// TIA Portal V18 export
FUNCTION "SS1_774A1_16DO_IO_Update" : Void   // FC11070, LAD
{ S7_Optimized_Access := 'TRUE' }
VERSION : 0.1
// stored: AutoNumber false, IsIECCheckEnabled false, SetENOAutomatically false, UDAEnableTagReadback false
BEGIN

REGION Network 1: DQa0
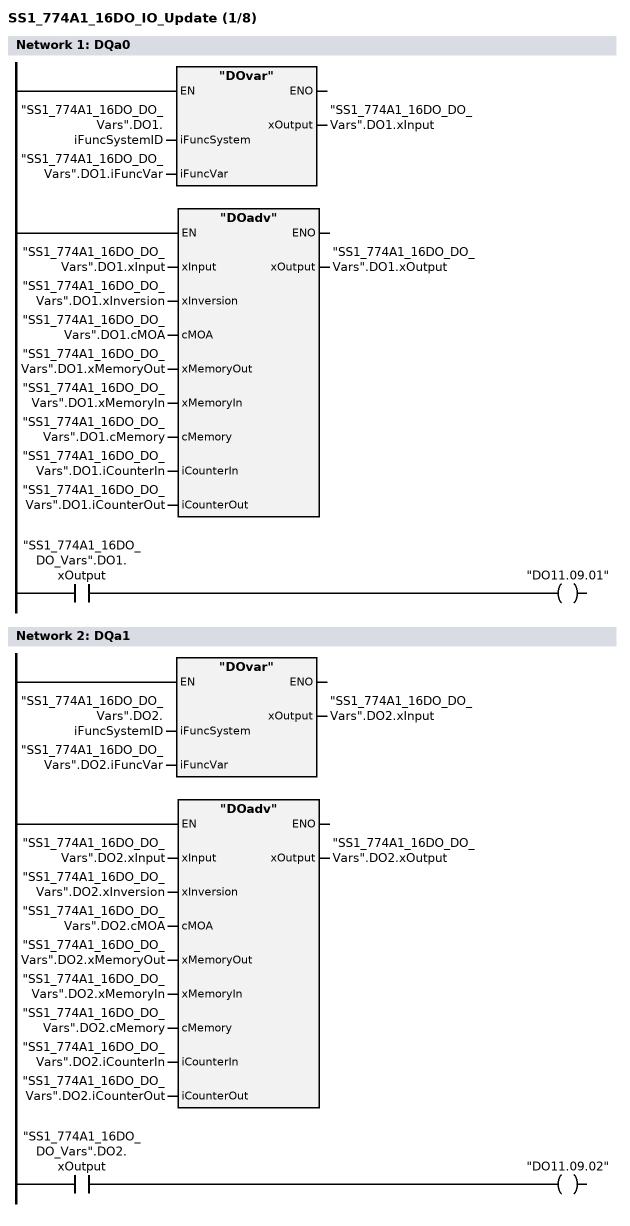
   RUNG wire#powerrail
      "DOvar"(iFuncSystem := "SS1_774A1_16DO_DO_Vars".DO1.iFuncSystemID, iFuncVar := "SS1_774A1_16DO_DO_Vars".DO1.iFuncVar, xOutput => "SS1_774A1_16DO_DO_Vars".DO1.xInput)
   END_RUNG
   RUNG wire#powerrail
      "DOadv"(xInput := "SS1_774A1_16DO_DO_Vars".DO1.xInput, xInversion := "SS1_774A1_16DO_DO_Vars".DO1.xInversion, cMOA := "SS1_774A1_16DO_DO_Vars".DO1.cMOA, xMemoryOut := "SS1_774A1_16DO_DO_Vars".DO1.xMemoryOut, xMemoryIn := "SS1_774A1_16DO_DO_Vars".DO1.xMemoryIn, cMemory := "SS1_774A1_16DO_DO_Vars".DO1.cMemory, iCounterIn := "SS1_774A1_16DO_DO_Vars".DO1.iCounterIn, iCounterOut := "SS1_774A1_16DO_DO_Vars".DO1.iCounterOut, xOutput => "SS1_774A1_16DO_DO_Vars".DO1.xOutput)
   END_RUNG
   RUNG wire#powerrail
      Contact( "SS1_774A1_16DO_DO_Vars".DO1.xOutput )
      Coil( "DO11.09.01" )
   END_RUNG
   // the same network as SCL:
   "DOvar"(iFuncSystem := "SS1_774A1_16DO_DO_Vars".DO1.iFuncSystemID,
           iFuncVar := "SS1_774A1_16DO_DO_Vars".DO1.iFuncVar,
           xOutput => "SS1_774A1_16DO_DO_Vars".DO1.xInput);
   "DOadv"(xInput := "SS1_774A1_16DO_DO_Vars".DO1.xInput,
           xInversion := "SS1_774A1_16DO_DO_Vars".DO1.xInversion,
           cMOA := "SS1_774A1_16DO_DO_Vars".DO1.cMOA,
           xMemoryOut := "SS1_774A1_16DO_DO_Vars".DO1.xMemoryOut,
           xMemoryIn := "SS1_774A1_16DO_DO_Vars".DO1.xMemoryIn,
           cMemory := "SS1_774A1_16DO_DO_Vars".DO1.cMemory,
           iCounterIn := "SS1_774A1_16DO_DO_Vars".DO1.iCounterIn,
           iCounterOut := "SS1_774A1_16DO_DO_Vars".DO1.iCounterOut,
           xOutput => "SS1_774A1_16DO_DO_Vars".DO1.xOutput);
   "DO11.09.01" := "SS1_774A1_16DO_DO_Vars".DO1.xOutput;
END_REGION

REGION Network 2: DQa1
   RUNG wire#powerrail
      "DOvar"(iFuncSystem := "SS1_774A1_16DO_DO_Vars".DO2.iFuncSystemID, iFuncVar := "SS1_774A1_16DO_DO_Vars".DO2.iFuncVar, xOutput => "SS1_774A1_16DO_DO_Vars".DO2.xInput)
   END_RUNG
   RUNG wire#powerrail
      "DOadv"(xInput := "SS1_774A1_16DO_DO_Vars".DO2.xInput, xInversion := "SS1_774A1_16DO_DO_Vars".DO2.xInversion, cMOA := "SS1_774A1_16DO_DO_Vars".DO2.cMOA, xMemoryOut := "SS1_774A1_16DO_DO_Vars".DO2.xMemoryOut, xMemoryIn := "SS1_774A1_16DO_DO_Vars".DO2.xMemoryIn, cMemory := "SS1_774A1_16DO_DO_Vars".DO2.cMemory, iCounterIn := "SS1_774A1_16DO_DO_Vars".DO2.iCounterIn, iCounterOut := "SS1_774A1_16DO_DO_Vars".DO2.iCounterOut, xOutput => "SS1_774A1_16DO_DO_Vars".DO2.xOutput)
   END_RUNG
   RUNG wire#powerrail
      Contact( "SS1_774A1_16DO_DO_Vars".DO2.xOutput )
      Coil( "DO11.09.02" )
   END_RUNG
   // the same network as SCL:
   "DOvar"(iFuncSystem := "SS1_774A1_16DO_DO_Vars".DO2.iFuncSystemID,
           iFuncVar := "SS1_774A1_16DO_DO_Vars".DO2.iFuncVar,
           xOutput => "SS1_774A1_16DO_DO_Vars".DO2.xInput);
   "DOadv"(xInput := "SS1_774A1_16DO_DO_Vars".DO2.xInput,
           xInversion := "SS1_774A1_16DO_DO_Vars".DO2.xInversion,
           cMOA := "SS1_774A1_16DO_DO_Vars".DO2.cMOA,
           xMemoryOut := "SS1_774A1_16DO_DO_Vars".DO2.xMemoryOut,
           xMemoryIn := "SS1_774A1_16DO_DO_Vars".DO2.xMemoryIn,
           cMemory := "SS1_774A1_16DO_DO_Vars".DO2.cMemory,
           iCounterIn := "SS1_774A1_16DO_DO_Vars".DO2.iCounterIn,
           iCounterOut := "SS1_774A1_16DO_DO_Vars".DO2.iCounterOut,
           xOutput => "SS1_774A1_16DO_DO_Vars".DO2.xOutput);
   "DO11.09.02" := "SS1_774A1_16DO_DO_Vars".DO2.xOutput;
END_REGION

REGION Network 3: DQa2
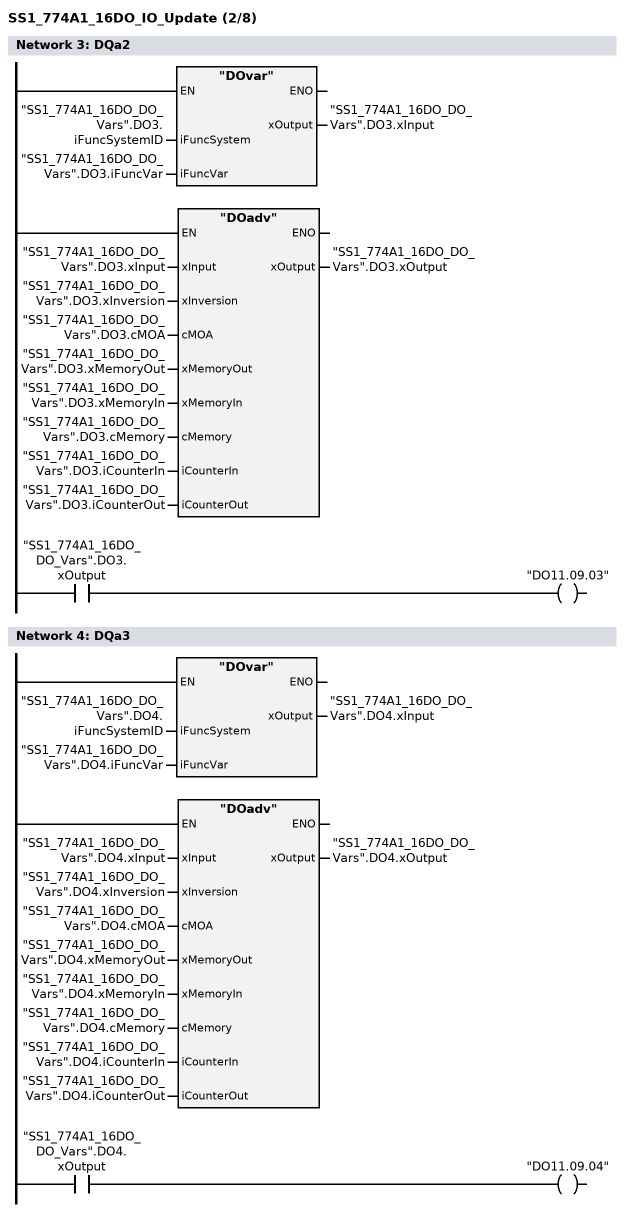
   RUNG wire#powerrail
      "DOvar"(iFuncSystem := "SS1_774A1_16DO_DO_Vars".DO3.iFuncSystemID, iFuncVar := "SS1_774A1_16DO_DO_Vars".DO3.iFuncVar, xOutput => "SS1_774A1_16DO_DO_Vars".DO3.xInput)
   END_RUNG
   RUNG wire#powerrail
      "DOadv"(xInput := "SS1_774A1_16DO_DO_Vars".DO3.xInput, xInversion := "SS1_774A1_16DO_DO_Vars".DO3.xInversion, cMOA := "SS1_774A1_16DO_DO_Vars".DO3.cMOA, xMemoryOut := "SS1_774A1_16DO_DO_Vars".DO3.xMemoryOut, xMemoryIn := "SS1_774A1_16DO_DO_Vars".DO3.xMemoryIn, cMemory := "SS1_774A1_16DO_DO_Vars".DO3.cMemory, iCounterIn := "SS1_774A1_16DO_DO_Vars".DO3.iCounterIn, iCounterOut := "SS1_774A1_16DO_DO_Vars".DO3.iCounterOut, xOutput => "SS1_774A1_16DO_DO_Vars".DO3.xOutput)
   END_RUNG
   RUNG wire#powerrail
      Contact( "SS1_774A1_16DO_DO_Vars".DO3.xOutput )
      Coil( "DO11.09.03" )
   END_RUNG
   // the same network as SCL:
   "DOvar"(iFuncSystem := "SS1_774A1_16DO_DO_Vars".DO3.iFuncSystemID,
           iFuncVar := "SS1_774A1_16DO_DO_Vars".DO3.iFuncVar,
           xOutput => "SS1_774A1_16DO_DO_Vars".DO3.xInput);
   "DOadv"(xInput := "SS1_774A1_16DO_DO_Vars".DO3.xInput,
           xInversion := "SS1_774A1_16DO_DO_Vars".DO3.xInversion,
           cMOA := "SS1_774A1_16DO_DO_Vars".DO3.cMOA,
           xMemoryOut := "SS1_774A1_16DO_DO_Vars".DO3.xMemoryOut,
           xMemoryIn := "SS1_774A1_16DO_DO_Vars".DO3.xMemoryIn,
           cMemory := "SS1_774A1_16DO_DO_Vars".DO3.cMemory,
           iCounterIn := "SS1_774A1_16DO_DO_Vars".DO3.iCounterIn,
           iCounterOut := "SS1_774A1_16DO_DO_Vars".DO3.iCounterOut,
           xOutput => "SS1_774A1_16DO_DO_Vars".DO3.xOutput);
   "DO11.09.03" := "SS1_774A1_16DO_DO_Vars".DO3.xOutput;
END_REGION

REGION Network 4: DQa3
   RUNG wire#powerrail
      "DOvar"(iFuncSystem := "SS1_774A1_16DO_DO_Vars".DO4.iFuncSystemID, iFuncVar := "SS1_774A1_16DO_DO_Vars".DO4.iFuncVar, xOutput => "SS1_774A1_16DO_DO_Vars".DO4.xInput)
   END_RUNG
   RUNG wire#powerrail
      "DOadv"(xInput := "SS1_774A1_16DO_DO_Vars".DO4.xInput, xInversion := "SS1_774A1_16DO_DO_Vars".DO4.xInversion, cMOA := "SS1_774A1_16DO_DO_Vars".DO4.cMOA, xMemoryOut := "SS1_774A1_16DO_DO_Vars".DO4.xMemoryOut, xMemoryIn := "SS1_774A1_16DO_DO_Vars".DO4.xMemoryIn, cMemory := "SS1_774A1_16DO_DO_Vars".DO4.cMemory, iCounterIn := "SS1_774A1_16DO_DO_Vars".DO4.iCounterIn, iCounterOut := "SS1_774A1_16DO_DO_Vars".DO4.iCounterOut, xOutput => "SS1_774A1_16DO_DO_Vars".DO4.xOutput)
   END_RUNG
   RUNG wire#powerrail
      Contact( "SS1_774A1_16DO_DO_Vars".DO4.xOutput )
      Coil( "DO11.09.04" )
   END_RUNG
   // the same network as SCL:
   "DOvar"(iFuncSystem := "SS1_774A1_16DO_DO_Vars".DO4.iFuncSystemID,
           iFuncVar := "SS1_774A1_16DO_DO_Vars".DO4.iFuncVar,
           xOutput => "SS1_774A1_16DO_DO_Vars".DO4.xInput);
   "DOadv"(xInput := "SS1_774A1_16DO_DO_Vars".DO4.xInput,
           xInversion := "SS1_774A1_16DO_DO_Vars".DO4.xInversion,
           cMOA := "SS1_774A1_16DO_DO_Vars".DO4.cMOA,
           xMemoryOut := "SS1_774A1_16DO_DO_Vars".DO4.xMemoryOut,
           xMemoryIn := "SS1_774A1_16DO_DO_Vars".DO4.xMemoryIn,
           cMemory := "SS1_774A1_16DO_DO_Vars".DO4.cMemory,
           iCounterIn := "SS1_774A1_16DO_DO_Vars".DO4.iCounterIn,
           iCounterOut := "SS1_774A1_16DO_DO_Vars".DO4.iCounterOut,
           xOutput => "SS1_774A1_16DO_DO_Vars".DO4.xOutput);
   "DO11.09.04" := "SS1_774A1_16DO_DO_Vars".DO4.xOutput;
END_REGION

REGION Network 5: DQa4
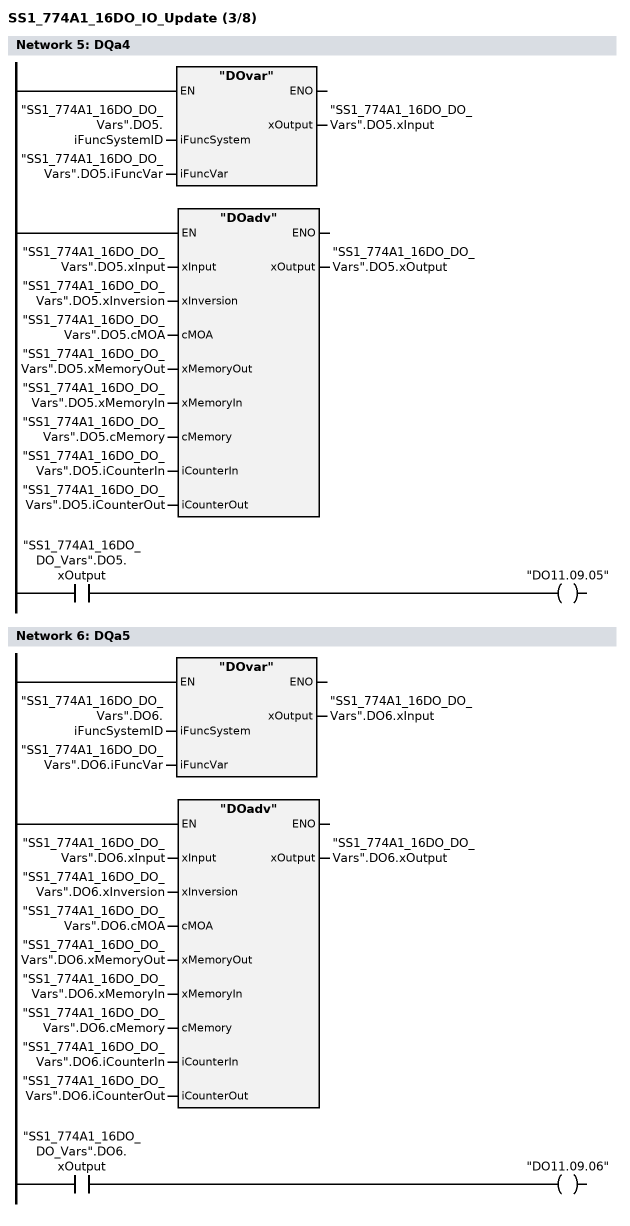
   RUNG wire#powerrail
      "DOvar"(iFuncSystem := "SS1_774A1_16DO_DO_Vars".DO5.iFuncSystemID, iFuncVar := "SS1_774A1_16DO_DO_Vars".DO5.iFuncVar, xOutput => "SS1_774A1_16DO_DO_Vars".DO5.xInput)
   END_RUNG
   RUNG wire#powerrail
      "DOadv"(xInput := "SS1_774A1_16DO_DO_Vars".DO5.xInput, xInversion := "SS1_774A1_16DO_DO_Vars".DO5.xInversion, cMOA := "SS1_774A1_16DO_DO_Vars".DO5.cMOA, xMemoryOut := "SS1_774A1_16DO_DO_Vars".DO5.xMemoryOut, xMemoryIn := "SS1_774A1_16DO_DO_Vars".DO5.xMemoryIn, cMemory := "SS1_774A1_16DO_DO_Vars".DO5.cMemory, iCounterIn := "SS1_774A1_16DO_DO_Vars".DO5.iCounterIn, iCounterOut := "SS1_774A1_16DO_DO_Vars".DO5.iCounterOut, xOutput => "SS1_774A1_16DO_DO_Vars".DO5.xOutput)
   END_RUNG
   RUNG wire#powerrail
      Contact( "SS1_774A1_16DO_DO_Vars".DO5.xOutput )
      Coil( "DO11.09.05" )
   END_RUNG
   // the same network as SCL:
   "DOvar"(iFuncSystem := "SS1_774A1_16DO_DO_Vars".DO5.iFuncSystemID,
           iFuncVar := "SS1_774A1_16DO_DO_Vars".DO5.iFuncVar,
           xOutput => "SS1_774A1_16DO_DO_Vars".DO5.xInput);
   "DOadv"(xInput := "SS1_774A1_16DO_DO_Vars".DO5.xInput,
           xInversion := "SS1_774A1_16DO_DO_Vars".DO5.xInversion,
           cMOA := "SS1_774A1_16DO_DO_Vars".DO5.cMOA,
           xMemoryOut := "SS1_774A1_16DO_DO_Vars".DO5.xMemoryOut,
           xMemoryIn := "SS1_774A1_16DO_DO_Vars".DO5.xMemoryIn,
           cMemory := "SS1_774A1_16DO_DO_Vars".DO5.cMemory,
           iCounterIn := "SS1_774A1_16DO_DO_Vars".DO5.iCounterIn,
           iCounterOut := "SS1_774A1_16DO_DO_Vars".DO5.iCounterOut,
           xOutput => "SS1_774A1_16DO_DO_Vars".DO5.xOutput);
   "DO11.09.05" := "SS1_774A1_16DO_DO_Vars".DO5.xOutput;
END_REGION

REGION Network 6: DQa5
   RUNG wire#powerrail
      "DOvar"(iFuncSystem := "SS1_774A1_16DO_DO_Vars".DO6.iFuncSystemID, iFuncVar := "SS1_774A1_16DO_DO_Vars".DO6.iFuncVar, xOutput => "SS1_774A1_16DO_DO_Vars".DO6.xInput)
   END_RUNG
   RUNG wire#powerrail
      "DOadv"(xInput := "SS1_774A1_16DO_DO_Vars".DO6.xInput, xInversion := "SS1_774A1_16DO_DO_Vars".DO6.xInversion, cMOA := "SS1_774A1_16DO_DO_Vars".DO6.cMOA, xMemoryOut := "SS1_774A1_16DO_DO_Vars".DO6.xMemoryOut, xMemoryIn := "SS1_774A1_16DO_DO_Vars".DO6.xMemoryIn, cMemory := "SS1_774A1_16DO_DO_Vars".DO6.cMemory, iCounterIn := "SS1_774A1_16DO_DO_Vars".DO6.iCounterIn, iCounterOut := "SS1_774A1_16DO_DO_Vars".DO6.iCounterOut, xOutput => "SS1_774A1_16DO_DO_Vars".DO6.xOutput)
   END_RUNG
   RUNG wire#powerrail
      Contact( "SS1_774A1_16DO_DO_Vars".DO6.xOutput )
      Coil( "DO11.09.06" )
   END_RUNG
   // the same network as SCL:
   "DOvar"(iFuncSystem := "SS1_774A1_16DO_DO_Vars".DO6.iFuncSystemID,
           iFuncVar := "SS1_774A1_16DO_DO_Vars".DO6.iFuncVar,
           xOutput => "SS1_774A1_16DO_DO_Vars".DO6.xInput);
   "DOadv"(xInput := "SS1_774A1_16DO_DO_Vars".DO6.xInput,
           xInversion := "SS1_774A1_16DO_DO_Vars".DO6.xInversion,
           cMOA := "SS1_774A1_16DO_DO_Vars".DO6.cMOA,
           xMemoryOut := "SS1_774A1_16DO_DO_Vars".DO6.xMemoryOut,
           xMemoryIn := "SS1_774A1_16DO_DO_Vars".DO6.xMemoryIn,
           cMemory := "SS1_774A1_16DO_DO_Vars".DO6.cMemory,
           iCounterIn := "SS1_774A1_16DO_DO_Vars".DO6.iCounterIn,
           iCounterOut := "SS1_774A1_16DO_DO_Vars".DO6.iCounterOut,
           xOutput => "SS1_774A1_16DO_DO_Vars".DO6.xOutput);
   "DO11.09.06" := "SS1_774A1_16DO_DO_Vars".DO6.xOutput;
END_REGION

REGION Network 7: DQa6
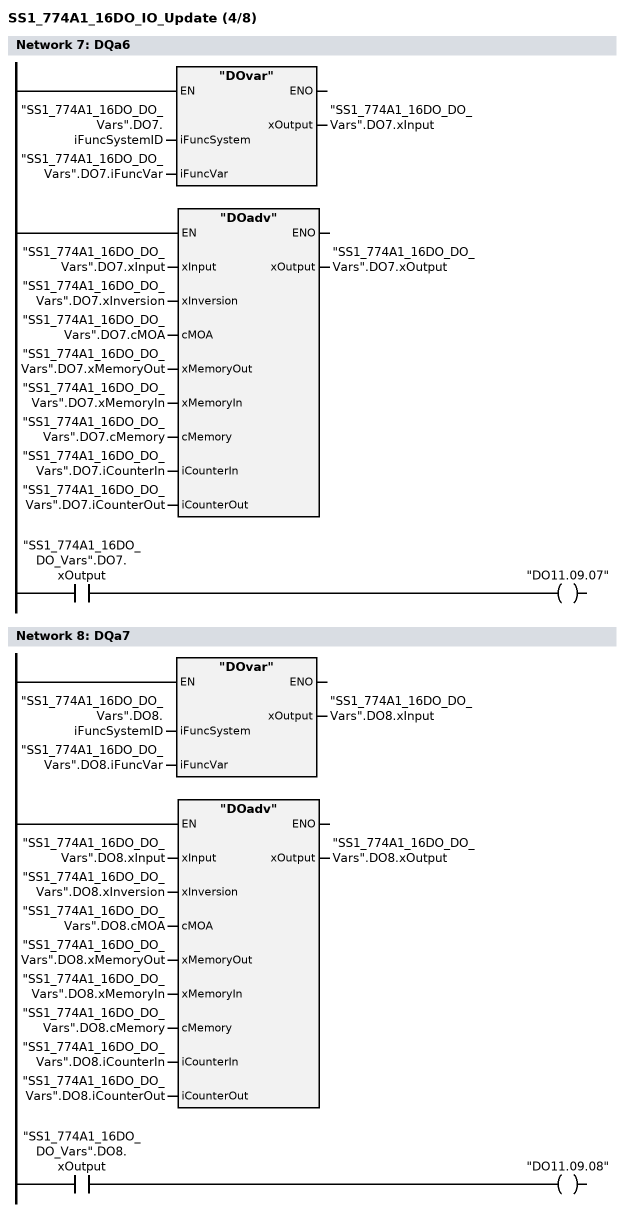
   RUNG wire#powerrail
      "DOvar"(iFuncSystem := "SS1_774A1_16DO_DO_Vars".DO7.iFuncSystemID, iFuncVar := "SS1_774A1_16DO_DO_Vars".DO7.iFuncVar, xOutput => "SS1_774A1_16DO_DO_Vars".DO7.xInput)
   END_RUNG
   RUNG wire#powerrail
      "DOadv"(xInput := "SS1_774A1_16DO_DO_Vars".DO7.xInput, xInversion := "SS1_774A1_16DO_DO_Vars".DO7.xInversion, cMOA := "SS1_774A1_16DO_DO_Vars".DO7.cMOA, xMemoryOut := "SS1_774A1_16DO_DO_Vars".DO7.xMemoryOut, xMemoryIn := "SS1_774A1_16DO_DO_Vars".DO7.xMemoryIn, cMemory := "SS1_774A1_16DO_DO_Vars".DO7.cMemory, iCounterIn := "SS1_774A1_16DO_DO_Vars".DO7.iCounterIn, iCounterOut := "SS1_774A1_16DO_DO_Vars".DO7.iCounterOut, xOutput => "SS1_774A1_16DO_DO_Vars".DO7.xOutput)
   END_RUNG
   RUNG wire#powerrail
      Contact( "SS1_774A1_16DO_DO_Vars".DO7.xOutput )
      Coil( "DO11.09.07" )
   END_RUNG
   // the same network as SCL:
   "DOvar"(iFuncSystem := "SS1_774A1_16DO_DO_Vars".DO7.iFuncSystemID,
           iFuncVar := "SS1_774A1_16DO_DO_Vars".DO7.iFuncVar,
           xOutput => "SS1_774A1_16DO_DO_Vars".DO7.xInput);
   "DOadv"(xInput := "SS1_774A1_16DO_DO_Vars".DO7.xInput,
           xInversion := "SS1_774A1_16DO_DO_Vars".DO7.xInversion,
           cMOA := "SS1_774A1_16DO_DO_Vars".DO7.cMOA,
           xMemoryOut := "SS1_774A1_16DO_DO_Vars".DO7.xMemoryOut,
           xMemoryIn := "SS1_774A1_16DO_DO_Vars".DO7.xMemoryIn,
           cMemory := "SS1_774A1_16DO_DO_Vars".DO7.cMemory,
           iCounterIn := "SS1_774A1_16DO_DO_Vars".DO7.iCounterIn,
           iCounterOut := "SS1_774A1_16DO_DO_Vars".DO7.iCounterOut,
           xOutput => "SS1_774A1_16DO_DO_Vars".DO7.xOutput);
   "DO11.09.07" := "SS1_774A1_16DO_DO_Vars".DO7.xOutput;
END_REGION

REGION Network 8: DQa7
   RUNG wire#powerrail
      "DOvar"(iFuncSystem := "SS1_774A1_16DO_DO_Vars".DO8.iFuncSystemID, iFuncVar := "SS1_774A1_16DO_DO_Vars".DO8.iFuncVar, xOutput => "SS1_774A1_16DO_DO_Vars".DO8.xInput)
   END_RUNG
   RUNG wire#powerrail
      "DOadv"(xInput := "SS1_774A1_16DO_DO_Vars".DO8.xInput, xInversion := "SS1_774A1_16DO_DO_Vars".DO8.xInversion, cMOA := "SS1_774A1_16DO_DO_Vars".DO8.cMOA, xMemoryOut := "SS1_774A1_16DO_DO_Vars".DO8.xMemoryOut, xMemoryIn := "SS1_774A1_16DO_DO_Vars".DO8.xMemoryIn, cMemory := "SS1_774A1_16DO_DO_Vars".DO8.cMemory, iCounterIn := "SS1_774A1_16DO_DO_Vars".DO8.iCounterIn, iCounterOut := "SS1_774A1_16DO_DO_Vars".DO8.iCounterOut, xOutput => "SS1_774A1_16DO_DO_Vars".DO8.xOutput)
   END_RUNG
   RUNG wire#powerrail
      Contact( "SS1_774A1_16DO_DO_Vars".DO8.xOutput )
      Coil( "DO11.09.08" )
   END_RUNG
   // the same network as SCL:
   "DOvar"(iFuncSystem := "SS1_774A1_16DO_DO_Vars".DO8.iFuncSystemID,
           iFuncVar := "SS1_774A1_16DO_DO_Vars".DO8.iFuncVar,
           xOutput => "SS1_774A1_16DO_DO_Vars".DO8.xInput);
   "DOadv"(xInput := "SS1_774A1_16DO_DO_Vars".DO8.xInput,
           xInversion := "SS1_774A1_16DO_DO_Vars".DO8.xInversion,
           cMOA := "SS1_774A1_16DO_DO_Vars".DO8.cMOA,
           xMemoryOut := "SS1_774A1_16DO_DO_Vars".DO8.xMemoryOut,
           xMemoryIn := "SS1_774A1_16DO_DO_Vars".DO8.xMemoryIn,
           cMemory := "SS1_774A1_16DO_DO_Vars".DO8.cMemory,
           iCounterIn := "SS1_774A1_16DO_DO_Vars".DO8.iCounterIn,
           iCounterOut := "SS1_774A1_16DO_DO_Vars".DO8.iCounterOut,
           xOutput => "SS1_774A1_16DO_DO_Vars".DO8.xOutput);
   "DO11.09.08" := "SS1_774A1_16DO_DO_Vars".DO8.xOutput;
END_REGION

REGION Network 9: DQb0
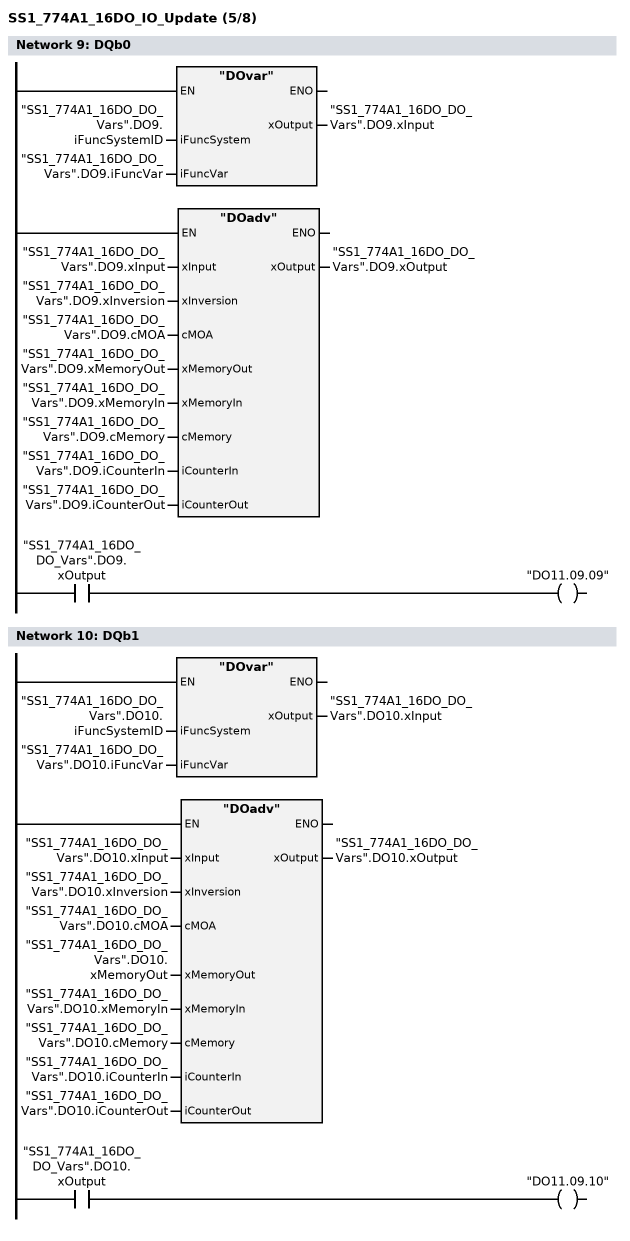
   RUNG wire#powerrail
      "DOvar"(iFuncSystem := "SS1_774A1_16DO_DO_Vars".DO9.iFuncSystemID, iFuncVar := "SS1_774A1_16DO_DO_Vars".DO9.iFuncVar, xOutput => "SS1_774A1_16DO_DO_Vars".DO9.xInput)
   END_RUNG
   RUNG wire#powerrail
      "DOadv"(xInput := "SS1_774A1_16DO_DO_Vars".DO9.xInput, xInversion := "SS1_774A1_16DO_DO_Vars".DO9.xInversion, cMOA := "SS1_774A1_16DO_DO_Vars".DO9.cMOA, xMemoryOut := "SS1_774A1_16DO_DO_Vars".DO9.xMemoryOut, xMemoryIn := "SS1_774A1_16DO_DO_Vars".DO9.xMemoryIn, cMemory := "SS1_774A1_16DO_DO_Vars".DO9.cMemory, iCounterIn := "SS1_774A1_16DO_DO_Vars".DO9.iCounterIn, iCounterOut := "SS1_774A1_16DO_DO_Vars".DO9.iCounterOut, xOutput => "SS1_774A1_16DO_DO_Vars".DO9.xOutput)
   END_RUNG
   RUNG wire#powerrail
      Contact( "SS1_774A1_16DO_DO_Vars".DO9.xOutput )
      Coil( "DO11.09.09" )
   END_RUNG
   // the same network as SCL:
   "DOvar"(iFuncSystem := "SS1_774A1_16DO_DO_Vars".DO9.iFuncSystemID,
           iFuncVar := "SS1_774A1_16DO_DO_Vars".DO9.iFuncVar,
           xOutput => "SS1_774A1_16DO_DO_Vars".DO9.xInput);
   "DOadv"(xInput := "SS1_774A1_16DO_DO_Vars".DO9.xInput,
           xInversion := "SS1_774A1_16DO_DO_Vars".DO9.xInversion,
           cMOA := "SS1_774A1_16DO_DO_Vars".DO9.cMOA,
           xMemoryOut := "SS1_774A1_16DO_DO_Vars".DO9.xMemoryOut,
           xMemoryIn := "SS1_774A1_16DO_DO_Vars".DO9.xMemoryIn,
           cMemory := "SS1_774A1_16DO_DO_Vars".DO9.cMemory,
           iCounterIn := "SS1_774A1_16DO_DO_Vars".DO9.iCounterIn,
           iCounterOut := "SS1_774A1_16DO_DO_Vars".DO9.iCounterOut,
           xOutput => "SS1_774A1_16DO_DO_Vars".DO9.xOutput);
   "DO11.09.09" := "SS1_774A1_16DO_DO_Vars".DO9.xOutput;
END_REGION

REGION Network 10: DQb1
   RUNG wire#powerrail
      "DOvar"(iFuncSystem := "SS1_774A1_16DO_DO_Vars".DO10.iFuncSystemID, iFuncVar := "SS1_774A1_16DO_DO_Vars".DO10.iFuncVar, xOutput => "SS1_774A1_16DO_DO_Vars".DO10.xInput)
   END_RUNG
   RUNG wire#powerrail
      "DOadv"(xInput := "SS1_774A1_16DO_DO_Vars".DO10.xInput, xInversion := "SS1_774A1_16DO_DO_Vars".DO10.xInversion, cMOA := "SS1_774A1_16DO_DO_Vars".DO10.cMOA, xMemoryOut := "SS1_774A1_16DO_DO_Vars".DO10.xMemoryOut, xMemoryIn := "SS1_774A1_16DO_DO_Vars".DO10.xMemoryIn, cMemory := "SS1_774A1_16DO_DO_Vars".DO10.cMemory, iCounterIn := "SS1_774A1_16DO_DO_Vars".DO10.iCounterIn, iCounterOut := "SS1_774A1_16DO_DO_Vars".DO10.iCounterOut, xOutput => "SS1_774A1_16DO_DO_Vars".DO10.xOutput)
   END_RUNG
   RUNG wire#powerrail
      Contact( "SS1_774A1_16DO_DO_Vars".DO10.xOutput )
      Coil( "DO11.09.10" )
   END_RUNG
   // the same network as SCL:
   "DOvar"(iFuncSystem := "SS1_774A1_16DO_DO_Vars".DO10.iFuncSystemID,
           iFuncVar := "SS1_774A1_16DO_DO_Vars".DO10.iFuncVar,
           xOutput => "SS1_774A1_16DO_DO_Vars".DO10.xInput);
   "DOadv"(xInput := "SS1_774A1_16DO_DO_Vars".DO10.xInput,
           xInversion := "SS1_774A1_16DO_DO_Vars".DO10.xInversion,
           cMOA := "SS1_774A1_16DO_DO_Vars".DO10.cMOA,
           xMemoryOut := "SS1_774A1_16DO_DO_Vars".DO10.xMemoryOut,
           xMemoryIn := "SS1_774A1_16DO_DO_Vars".DO10.xMemoryIn,
           cMemory := "SS1_774A1_16DO_DO_Vars".DO10.cMemory,
           iCounterIn := "SS1_774A1_16DO_DO_Vars".DO10.iCounterIn,
           iCounterOut := "SS1_774A1_16DO_DO_Vars".DO10.iCounterOut,
           xOutput => "SS1_774A1_16DO_DO_Vars".DO10.xOutput);
   "DO11.09.10" := "SS1_774A1_16DO_DO_Vars".DO10.xOutput;
END_REGION

REGION Network 11: DQb2
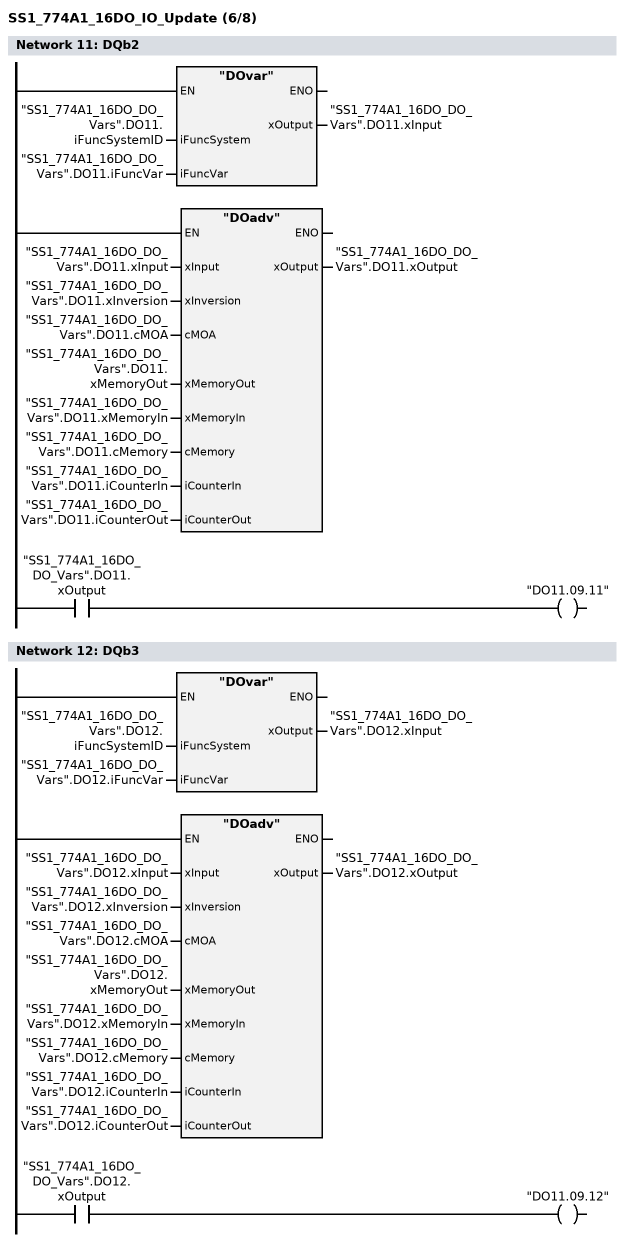
   RUNG wire#powerrail
      "DOvar"(iFuncSystem := "SS1_774A1_16DO_DO_Vars".DO11.iFuncSystemID, iFuncVar := "SS1_774A1_16DO_DO_Vars".DO11.iFuncVar, xOutput => "SS1_774A1_16DO_DO_Vars".DO11.xInput)
   END_RUNG
   RUNG wire#powerrail
      "DOadv"(xInput := "SS1_774A1_16DO_DO_Vars".DO11.xInput, xInversion := "SS1_774A1_16DO_DO_Vars".DO11.xInversion, cMOA := "SS1_774A1_16DO_DO_Vars".DO11.cMOA, xMemoryOut := "SS1_774A1_16DO_DO_Vars".DO11.xMemoryOut, xMemoryIn := "SS1_774A1_16DO_DO_Vars".DO11.xMemoryIn, cMemory := "SS1_774A1_16DO_DO_Vars".DO11.cMemory, iCounterIn := "SS1_774A1_16DO_DO_Vars".DO11.iCounterIn, iCounterOut := "SS1_774A1_16DO_DO_Vars".DO11.iCounterOut, xOutput => "SS1_774A1_16DO_DO_Vars".DO11.xOutput)
   END_RUNG
   RUNG wire#powerrail
      Contact( "SS1_774A1_16DO_DO_Vars".DO11.xOutput )
      Coil( "DO11.09.11" )
   END_RUNG
   // the same network as SCL:
   "DOvar"(iFuncSystem := "SS1_774A1_16DO_DO_Vars".DO11.iFuncSystemID,
           iFuncVar := "SS1_774A1_16DO_DO_Vars".DO11.iFuncVar,
           xOutput => "SS1_774A1_16DO_DO_Vars".DO11.xInput);
   "DOadv"(xInput := "SS1_774A1_16DO_DO_Vars".DO11.xInput,
           xInversion := "SS1_774A1_16DO_DO_Vars".DO11.xInversion,
           cMOA := "SS1_774A1_16DO_DO_Vars".DO11.cMOA,
           xMemoryOut := "SS1_774A1_16DO_DO_Vars".DO11.xMemoryOut,
           xMemoryIn := "SS1_774A1_16DO_DO_Vars".DO11.xMemoryIn,
           cMemory := "SS1_774A1_16DO_DO_Vars".DO11.cMemory,
           iCounterIn := "SS1_774A1_16DO_DO_Vars".DO11.iCounterIn,
           iCounterOut := "SS1_774A1_16DO_DO_Vars".DO11.iCounterOut,
           xOutput => "SS1_774A1_16DO_DO_Vars".DO11.xOutput);
   "DO11.09.11" := "SS1_774A1_16DO_DO_Vars".DO11.xOutput;
END_REGION

REGION Network 12: DQb3
   RUNG wire#powerrail
      "DOvar"(iFuncSystem := "SS1_774A1_16DO_DO_Vars".DO12.iFuncSystemID, iFuncVar := "SS1_774A1_16DO_DO_Vars".DO12.iFuncVar, xOutput => "SS1_774A1_16DO_DO_Vars".DO12.xInput)
   END_RUNG
   RUNG wire#powerrail
      "DOadv"(xInput := "SS1_774A1_16DO_DO_Vars".DO12.xInput, xInversion := "SS1_774A1_16DO_DO_Vars".DO12.xInversion, cMOA := "SS1_774A1_16DO_DO_Vars".DO12.cMOA, xMemoryOut := "SS1_774A1_16DO_DO_Vars".DO12.xMemoryOut, xMemoryIn := "SS1_774A1_16DO_DO_Vars".DO12.xMemoryIn, cMemory := "SS1_774A1_16DO_DO_Vars".DO12.cMemory, iCounterIn := "SS1_774A1_16DO_DO_Vars".DO12.iCounterIn, iCounterOut := "SS1_774A1_16DO_DO_Vars".DO12.iCounterOut, xOutput => "SS1_774A1_16DO_DO_Vars".DO12.xOutput)
   END_RUNG
   RUNG wire#powerrail
      Contact( "SS1_774A1_16DO_DO_Vars".DO12.xOutput )
      Coil( "DO11.09.12" )
   END_RUNG
   // the same network as SCL:
   "DOvar"(iFuncSystem := "SS1_774A1_16DO_DO_Vars".DO12.iFuncSystemID,
           iFuncVar := "SS1_774A1_16DO_DO_Vars".DO12.iFuncVar,
           xOutput => "SS1_774A1_16DO_DO_Vars".DO12.xInput);
   "DOadv"(xInput := "SS1_774A1_16DO_DO_Vars".DO12.xInput,
           xInversion := "SS1_774A1_16DO_DO_Vars".DO12.xInversion,
           cMOA := "SS1_774A1_16DO_DO_Vars".DO12.cMOA,
           xMemoryOut := "SS1_774A1_16DO_DO_Vars".DO12.xMemoryOut,
           xMemoryIn := "SS1_774A1_16DO_DO_Vars".DO12.xMemoryIn,
           cMemory := "SS1_774A1_16DO_DO_Vars".DO12.cMemory,
           iCounterIn := "SS1_774A1_16DO_DO_Vars".DO12.iCounterIn,
           iCounterOut := "SS1_774A1_16DO_DO_Vars".DO12.iCounterOut,
           xOutput => "SS1_774A1_16DO_DO_Vars".DO12.xOutput);
   "DO11.09.12" := "SS1_774A1_16DO_DO_Vars".DO12.xOutput;
END_REGION

REGION Network 13: DQb4
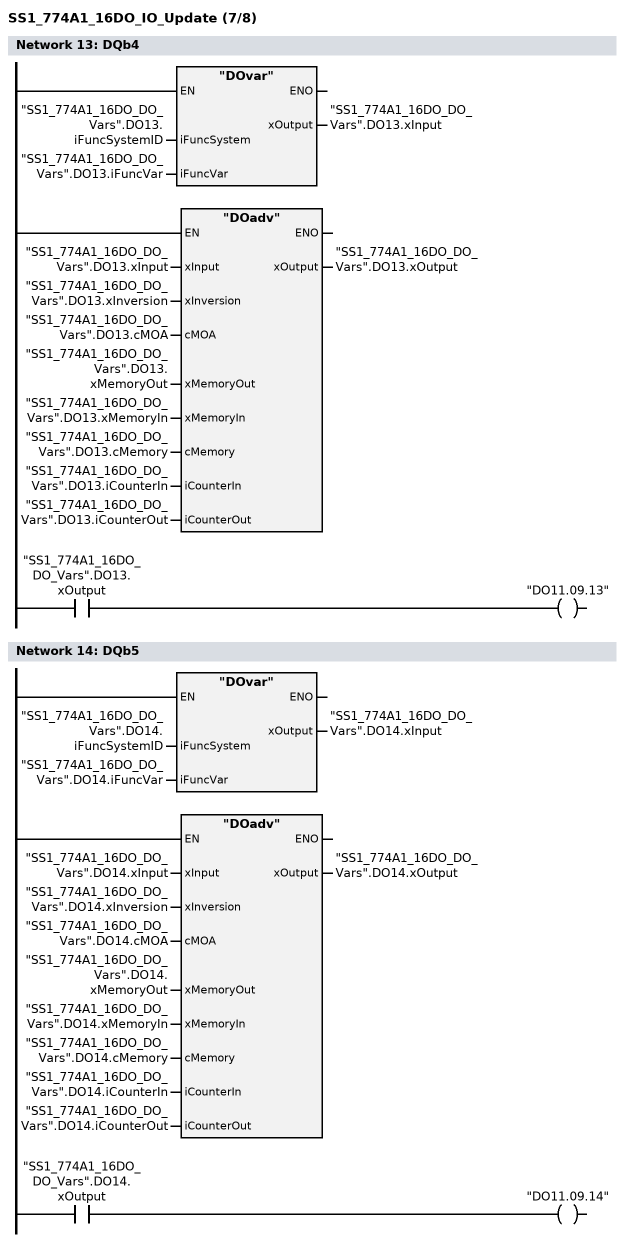
   RUNG wire#powerrail
      "DOvar"(iFuncSystem := "SS1_774A1_16DO_DO_Vars".DO13.iFuncSystemID, iFuncVar := "SS1_774A1_16DO_DO_Vars".DO13.iFuncVar, xOutput => "SS1_774A1_16DO_DO_Vars".DO13.xInput)
   END_RUNG
   RUNG wire#powerrail
      "DOadv"(xInput := "SS1_774A1_16DO_DO_Vars".DO13.xInput, xInversion := "SS1_774A1_16DO_DO_Vars".DO13.xInversion, cMOA := "SS1_774A1_16DO_DO_Vars".DO13.cMOA, xMemoryOut := "SS1_774A1_16DO_DO_Vars".DO13.xMemoryOut, xMemoryIn := "SS1_774A1_16DO_DO_Vars".DO13.xMemoryIn, cMemory := "SS1_774A1_16DO_DO_Vars".DO13.cMemory, iCounterIn := "SS1_774A1_16DO_DO_Vars".DO13.iCounterIn, iCounterOut := "SS1_774A1_16DO_DO_Vars".DO13.iCounterOut, xOutput => "SS1_774A1_16DO_DO_Vars".DO13.xOutput)
   END_RUNG
   RUNG wire#powerrail
      Contact( "SS1_774A1_16DO_DO_Vars".DO13.xOutput )
      Coil( "DO11.09.13" )
   END_RUNG
   // the same network as SCL:
   "DOvar"(iFuncSystem := "SS1_774A1_16DO_DO_Vars".DO13.iFuncSystemID,
           iFuncVar := "SS1_774A1_16DO_DO_Vars".DO13.iFuncVar,
           xOutput => "SS1_774A1_16DO_DO_Vars".DO13.xInput);
   "DOadv"(xInput := "SS1_774A1_16DO_DO_Vars".DO13.xInput,
           xInversion := "SS1_774A1_16DO_DO_Vars".DO13.xInversion,
           cMOA := "SS1_774A1_16DO_DO_Vars".DO13.cMOA,
           xMemoryOut := "SS1_774A1_16DO_DO_Vars".DO13.xMemoryOut,
           xMemoryIn := "SS1_774A1_16DO_DO_Vars".DO13.xMemoryIn,
           cMemory := "SS1_774A1_16DO_DO_Vars".DO13.cMemory,
           iCounterIn := "SS1_774A1_16DO_DO_Vars".DO13.iCounterIn,
           iCounterOut := "SS1_774A1_16DO_DO_Vars".DO13.iCounterOut,
           xOutput => "SS1_774A1_16DO_DO_Vars".DO13.xOutput);
   "DO11.09.13" := "SS1_774A1_16DO_DO_Vars".DO13.xOutput;
END_REGION

REGION Network 14: DQb5
   RUNG wire#powerrail
      "DOvar"(iFuncSystem := "SS1_774A1_16DO_DO_Vars".DO14.iFuncSystemID, iFuncVar := "SS1_774A1_16DO_DO_Vars".DO14.iFuncVar, xOutput => "SS1_774A1_16DO_DO_Vars".DO14.xInput)
   END_RUNG
   RUNG wire#powerrail
      "DOadv"(xInput := "SS1_774A1_16DO_DO_Vars".DO14.xInput, xInversion := "SS1_774A1_16DO_DO_Vars".DO14.xInversion, cMOA := "SS1_774A1_16DO_DO_Vars".DO14.cMOA, xMemoryOut := "SS1_774A1_16DO_DO_Vars".DO14.xMemoryOut, xMemoryIn := "SS1_774A1_16DO_DO_Vars".DO14.xMemoryIn, cMemory := "SS1_774A1_16DO_DO_Vars".DO14.cMemory, iCounterIn := "SS1_774A1_16DO_DO_Vars".DO14.iCounterIn, iCounterOut := "SS1_774A1_16DO_DO_Vars".DO14.iCounterOut, xOutput => "SS1_774A1_16DO_DO_Vars".DO14.xOutput)
   END_RUNG
   RUNG wire#powerrail
      Contact( "SS1_774A1_16DO_DO_Vars".DO14.xOutput )
      Coil( "DO11.09.14" )
   END_RUNG
   // the same network as SCL:
   "DOvar"(iFuncSystem := "SS1_774A1_16DO_DO_Vars".DO14.iFuncSystemID,
           iFuncVar := "SS1_774A1_16DO_DO_Vars".DO14.iFuncVar,
           xOutput => "SS1_774A1_16DO_DO_Vars".DO14.xInput);
   "DOadv"(xInput := "SS1_774A1_16DO_DO_Vars".DO14.xInput,
           xInversion := "SS1_774A1_16DO_DO_Vars".DO14.xInversion,
           cMOA := "SS1_774A1_16DO_DO_Vars".DO14.cMOA,
           xMemoryOut := "SS1_774A1_16DO_DO_Vars".DO14.xMemoryOut,
           xMemoryIn := "SS1_774A1_16DO_DO_Vars".DO14.xMemoryIn,
           cMemory := "SS1_774A1_16DO_DO_Vars".DO14.cMemory,
           iCounterIn := "SS1_774A1_16DO_DO_Vars".DO14.iCounterIn,
           iCounterOut := "SS1_774A1_16DO_DO_Vars".DO14.iCounterOut,
           xOutput => "SS1_774A1_16DO_DO_Vars".DO14.xOutput);
   "DO11.09.14" := "SS1_774A1_16DO_DO_Vars".DO14.xOutput;
END_REGION

REGION Network 15: DQb6
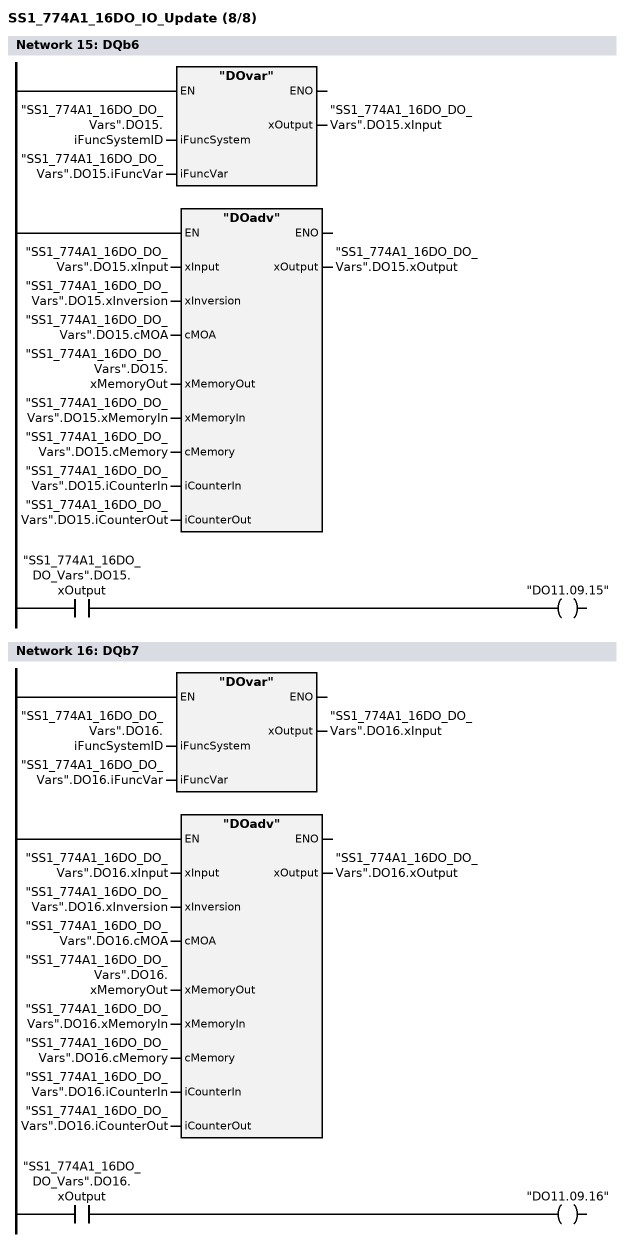
   RUNG wire#powerrail
      "DOvar"(iFuncSystem := "SS1_774A1_16DO_DO_Vars".DO15.iFuncSystemID, iFuncVar := "SS1_774A1_16DO_DO_Vars".DO15.iFuncVar, xOutput => "SS1_774A1_16DO_DO_Vars".DO15.xInput)
   END_RUNG
   RUNG wire#powerrail
      "DOadv"(xInput := "SS1_774A1_16DO_DO_Vars".DO15.xInput, xInversion := "SS1_774A1_16DO_DO_Vars".DO15.xInversion, cMOA := "SS1_774A1_16DO_DO_Vars".DO15.cMOA, xMemoryOut := "SS1_774A1_16DO_DO_Vars".DO15.xMemoryOut, xMemoryIn := "SS1_774A1_16DO_DO_Vars".DO15.xMemoryIn, cMemory := "SS1_774A1_16DO_DO_Vars".DO15.cMemory, iCounterIn := "SS1_774A1_16DO_DO_Vars".DO15.iCounterIn, iCounterOut := "SS1_774A1_16DO_DO_Vars".DO15.iCounterOut, xOutput => "SS1_774A1_16DO_DO_Vars".DO15.xOutput)
   END_RUNG
   RUNG wire#powerrail
      Contact( "SS1_774A1_16DO_DO_Vars".DO15.xOutput )
      Coil( "DO11.09.15" )
   END_RUNG
   // the same network as SCL:
   "DOvar"(iFuncSystem := "SS1_774A1_16DO_DO_Vars".DO15.iFuncSystemID,
           iFuncVar := "SS1_774A1_16DO_DO_Vars".DO15.iFuncVar,
           xOutput => "SS1_774A1_16DO_DO_Vars".DO15.xInput);
   "DOadv"(xInput := "SS1_774A1_16DO_DO_Vars".DO15.xInput,
           xInversion := "SS1_774A1_16DO_DO_Vars".DO15.xInversion,
           cMOA := "SS1_774A1_16DO_DO_Vars".DO15.cMOA,
           xMemoryOut := "SS1_774A1_16DO_DO_Vars".DO15.xMemoryOut,
           xMemoryIn := "SS1_774A1_16DO_DO_Vars".DO15.xMemoryIn,
           cMemory := "SS1_774A1_16DO_DO_Vars".DO15.cMemory,
           iCounterIn := "SS1_774A1_16DO_DO_Vars".DO15.iCounterIn,
           iCounterOut := "SS1_774A1_16DO_DO_Vars".DO15.iCounterOut,
           xOutput => "SS1_774A1_16DO_DO_Vars".DO15.xOutput);
   "DO11.09.15" := "SS1_774A1_16DO_DO_Vars".DO15.xOutput;
END_REGION

REGION Network 16: DQb7
   RUNG wire#powerrail
      "DOvar"(iFuncSystem := "SS1_774A1_16DO_DO_Vars".DO16.iFuncSystemID, iFuncVar := "SS1_774A1_16DO_DO_Vars".DO16.iFuncVar, xOutput => "SS1_774A1_16DO_DO_Vars".DO16.xInput)
   END_RUNG
   RUNG wire#powerrail
      "DOadv"(xInput := "SS1_774A1_16DO_DO_Vars".DO16.xInput, xInversion := "SS1_774A1_16DO_DO_Vars".DO16.xInversion, cMOA := "SS1_774A1_16DO_DO_Vars".DO16.cMOA, xMemoryOut := "SS1_774A1_16DO_DO_Vars".DO16.xMemoryOut, xMemoryIn := "SS1_774A1_16DO_DO_Vars".DO16.xMemoryIn, cMemory := "SS1_774A1_16DO_DO_Vars".DO16.cMemory, iCounterIn := "SS1_774A1_16DO_DO_Vars".DO16.iCounterIn, iCounterOut := "SS1_774A1_16DO_DO_Vars".DO16.iCounterOut, xOutput => "SS1_774A1_16DO_DO_Vars".DO16.xOutput)
   END_RUNG
   RUNG wire#powerrail
      Contact( "SS1_774A1_16DO_DO_Vars".DO16.xOutput )
      Coil( "DO11.09.16" )
   END_RUNG
   // the same network as SCL:
   "DOvar"(iFuncSystem := "SS1_774A1_16DO_DO_Vars".DO16.iFuncSystemID,
           iFuncVar := "SS1_774A1_16DO_DO_Vars".DO16.iFuncVar,
           xOutput => "SS1_774A1_16DO_DO_Vars".DO16.xInput);
   "DOadv"(xInput := "SS1_774A1_16DO_DO_Vars".DO16.xInput,
           xInversion := "SS1_774A1_16DO_DO_Vars".DO16.xInversion,
           cMOA := "SS1_774A1_16DO_DO_Vars".DO16.cMOA,
           xMemoryOut := "SS1_774A1_16DO_DO_Vars".DO16.xMemoryOut,
           xMemoryIn := "SS1_774A1_16DO_DO_Vars".DO16.xMemoryIn,
           cMemory := "SS1_774A1_16DO_DO_Vars".DO16.cMemory,
           iCounterIn := "SS1_774A1_16DO_DO_Vars".DO16.iCounterIn,
           iCounterOut := "SS1_774A1_16DO_DO_Vars".DO16.iCounterOut,
           xOutput => "SS1_774A1_16DO_DO_Vars".DO16.xOutput);
   "DO11.09.16" := "SS1_774A1_16DO_DO_Vars".DO16.xOutput;
END_REGION
END_FUNCTION
